PROGRAM MAIN
VAR
	RobotArm			: FB_RobotArm;
//	RobotArm1Inputs 	: ST_Inputs;
//	RobotArm1Outputs 	: ST_Outputs;
	
//SerialIndex : INT:=1;
//Index : INT;


//LSTEPS   : INT;
//RSTEPS   : INT;

//START    : BOOL;
END_VAR

//RobotArm(ST_Inputs := RobotArm1Inputs, ST_Outputs := RobotArm1Outputs);

RobotArm();

END_PROGRAM

(* stored: Version 1.1.0.1, ProductVersion 3.1.4024.9
   POU MAIN: Id {c1ea7bfa-a36b-4e65-912f-71822f4091f2}, SpecialFunc None *)
